{attribute 'pack_mode' := '0'}
TYPE ST_PLCOutputs :
STRUCT
	Q0: BYTE;
	Q1: BYTE;
	Q2: BYTE;
	Q3: BYTE;
	Q4: BYTE;
	Q5: BYTE;
	Q6: BYTE;
	Q7: BYTE;
	Q8: BYTE;
	Q9: BYTE;
	Q10: BYTE;
	Q11: BYTE;
	Q12: BYTE;
	Q13: BYTE;
	Q14: BYTE;
	Q15: BYTE;
	Q16: BYTE;
	Q17: BYTE;
	Q18: BYTE;
	Q19: BYTE;
	Q20: BYTE;
	Q21: BYTE;
	Q22: BYTE;
	Q23: BYTE;
	Q24: BYTE;
	Q25: BYTE;
	Q26: BYTE;
	Q27: BYTE;
	Q28: BYTE;
	Q29: BYTE;
	Q30: BYTE;
	Q31: BYTE;
	Q32: BYTE;
	Q33: BYTE;
	Q34: BYTE;
	Q35: BYTE;
	Q36: BYTE;
	Q37: BYTE;
	Q38: BYTE;
	Q39: BYTE;
	Q40: BYTE;
	Q41: BYTE;
	Q42: BYTE;
	Q43: BYTE;
	Q44: BYTE;
	Q45: BYTE;
	Q46: BYTE;
	Q47: BYTE;
	Q48: BYTE;
	Q49: BYTE;
	Q50: BYTE;
	Q51: BYTE;
	Q52: BYTE;
	Q53: BYTE;
	Q54: BYTE;
	Q55: BYTE;
	Q56: BYTE;
	Q57: BYTE;
	Q58: BYTE;
	Q59: BYTE;
	Q60: BYTE;
	Q61: BYTE;
	Q62: BYTE;
	Q63: BYTE;
	Q64: BYTE;
	Q65: BYTE;
	Q66: BYTE;
	Q67: BYTE;
	Q68: BYTE;
	Q69: BYTE;
	Q70: BYTE;
	Q71: BYTE;
	Q72: BYTE;
	Q73: BYTE;
	Q74: BYTE;
	Q75: BYTE;
	Q76: BYTE;
	Q77: BYTE;
	Q78: BYTE;
	Q79: BYTE;
	Q80: BYTE;
	Q81: BYTE;
	Q82: BYTE;
	Q83: BYTE;
	Q84: BYTE;
	Q85: BYTE;
	Q86: BYTE;
	Q87: BYTE;
	Q88: BYTE;
	Q89: BYTE;
	Q90: BYTE;
	Q91: BYTE;
	Q92: BYTE;
	Q93: BYTE;
	Q94: BYTE;
	Q95: BYTE;
	Q96: BYTE;
	Q97: BYTE;
	Q98: BYTE;
	Q99: BYTE;
	Q100: BYTE;
	Q101: BYTE;
	Q102: BYTE;
	Q103: BYTE;
	Q104: BYTE;
	Q105: BYTE;
	Q106: BYTE;
	Q107: BYTE;
	Q108: BYTE;
	Q109: BYTE;
	Q110: BYTE;
	Q111: BYTE;
	Q112: BYTE;
	Q113: BYTE;
	Q114: BYTE;
	Q115: BYTE;
	Q116: BYTE;
	Q117: BYTE;
	Q118: BYTE;
	Q119: BYTE;
	Q120: BYTE;
	Q121: BYTE;
	Q122: BYTE;
	Q123: BYTE;
	Q124: BYTE;
	Q125: BYTE;
	Q126: BYTE;
	Q127: BYTE;
	Q128: BYTE;
	Q129: BYTE;
	Q130: BYTE;
	Q131: BYTE;
	Q132: BYTE;
	Q133: BYTE;
	Q134: BYTE;
	Q135: BYTE;
	Q136: BYTE;
	Q137: BYTE;
	Q138: BYTE;
	Q139: BYTE;
	Q140: BYTE;
	Q141: BYTE;
	Q142: BYTE;
	Q143: BYTE;
	Q144: BYTE;
	Q145: BYTE;
	Q146: BYTE;
	Q147: BYTE;
	Q148: BYTE;
	Q149: BYTE;
	Q150: BYTE;
	Q151: BYTE;
	Q152: BYTE;
	Q153: BYTE;
	Q154: BYTE;
	Q155: BYTE;
	Q156: BYTE;
	Q157: BYTE;
	Q158: BYTE;
	Q159: BYTE;
	Q160: BYTE;
	Q161: BYTE;
	Q162: BYTE;
	Q163: BYTE;
	Q164: BYTE;
	Q165: BYTE;
	Q166: BYTE;
	Q167: BYTE;
	Q168: BYTE;
	Q169: BYTE;
	Q170: BYTE;
	Q171: BYTE;
	Q172: BYTE;
	Q173: BYTE;
	Q174: BYTE;
	Q175: BYTE;
	Q176: BYTE;
	Q177: BYTE;
	Q178: BYTE;
	Q179: BYTE;
	Q180: BYTE;
	Q181: BYTE;
	Q182: BYTE;
	Q183: BYTE;
	Q184: BYTE;
	Q185: BYTE;
	Q186: BYTE;
	Q187: BYTE;
	Q188: BYTE;
	Q189: BYTE;
	Q190: BYTE;
	Q191: BYTE;
	Q192: BYTE;
	Q193: BYTE;
	Q194: BYTE;
	Q195: BYTE;
	Q196: BYTE;
	Q197: BYTE;
	Q198: BYTE;
	Q199: BYTE;
	Q200: BYTE;
	Q201: BYTE;
	Q202: BYTE;
	Q203: BYTE;
	Q204: BYTE;
	Q205: BYTE;
	Q206: BYTE;
	Q207: BYTE;
	Q208: BYTE;
	Q209: BYTE;
	Q210: BYTE;
	Q211: BYTE;
	Q212: BYTE;
	Q213: BYTE;
	Q214: BYTE;
	Q215: BYTE;
	Q216: BYTE;
	Q217: BYTE;
	Q218: BYTE;
	Q219: BYTE;
	Q220: BYTE;
	Q221: BYTE;
	Q222: BYTE;
	Q223: BYTE;
	Q224: BYTE;
	Q225: BYTE;
	Q226: BYTE;
	Q227: BYTE;
	Q228: BYTE;
	Q229: BYTE;
	Q230: BYTE;
	Q231: BYTE;
	Q232: BYTE;
	Q233: BYTE;
	Q234: BYTE;
	Q235: BYTE;
	Q236: BYTE;
	Q237: BYTE;
	Q238: BYTE;
	Q239: BYTE;
	Q240: BYTE;
	Q241: BYTE;
	Q242: BYTE;
	Q243: BYTE;
	Q244: BYTE;
	Q245: BYTE;
	Q246: BYTE;
	Q247: BYTE;
	Q248: BYTE;
	Q249: BYTE;
	Q250: BYTE;
	Q251: BYTE;
	Q252: BYTE;
	Q253: BYTE;
	Q254: BYTE;
	Q255: BYTE;
	Q256: BYTE;
	Q257: BYTE;
	Q258: BYTE;
	Q259: BYTE;
	Q260: BYTE;
	Q261: BYTE;
	Q262: BYTE;
	Q263: BYTE;
	Q264: BYTE;
	Q265: BYTE;
	Q266: BYTE;
	Q267: BYTE;
	Q268: BYTE;
	Q269: BYTE;
	Q270: BYTE;
	Q271: BYTE;
	Q272: BYTE;
	Q273: BYTE;
	Q274: BYTE;
	Q275: BYTE;
	Q276: BYTE;
	Q277: BYTE;
	Q278: BYTE;
	Q279: BYTE;
	Q280: BYTE;
	Q281: BYTE;
	Q282: BYTE;
	Q283: BYTE;
	Q284: BYTE;
	Q285: BYTE;
	Q286: BYTE;
	Q287: BYTE;
	Q288: BYTE;
	Q289: BYTE;
	Q290: BYTE;
	Q291: BYTE;
	Q292: BYTE;
	Q293: BYTE;
	Q294: BYTE;
	Q295: BYTE;
	Q296: BYTE;
	Q297: BYTE;
	Q298: BYTE;
	Q299: BYTE;
	Q300: BYTE;
	Q301: BYTE;
	Q302: BYTE;
	Q303: BYTE;
	Q304: BYTE;
	Q305: BYTE;
	Q306: BYTE;
	Q307: BYTE;
	Q308: BYTE;
	Q309: BYTE;
	Q310: BYTE;
	Q311: BYTE;
	Q312: BYTE;
	Q313: BYTE;
	Q314: BYTE;
	Q315: BYTE;
	Q316: BYTE;
	Q317: BYTE;
	Q318: BYTE;
	Q319: BYTE;
	Q320: BYTE;
	Q321: BYTE;
	Q322: BYTE;
	Q323: BYTE;
	Q324: BYTE;
	Q325: BYTE;
	Q326: BYTE;
	Q327: BYTE;
	Q328: BYTE;
	Q329: BYTE;
	Q330: BYTE;
	Q331: BYTE;
	Q332: BYTE;
	Q333: BYTE;
	Q334: BYTE;
	Q335: BYTE;
	Q336: BYTE;
	Q337: BYTE;
	Q338: BYTE;
	Q339: BYTE;
	Q340: BYTE;
	Q341: BYTE;
	Q342: BYTE;
	Q343: BYTE;
	Q344: BYTE;
	Q345: BYTE;
	Q346: BYTE;
	Q347: BYTE;
	Q348: BYTE;
	Q349: BYTE;
	Q350: BYTE;
	Q351: BYTE;
	Q352: BYTE;
	Q353: BYTE;
	Q354: BYTE;
	Q355: BYTE;
	Q356: BYTE;
	Q357: BYTE;
	Q358: BYTE;
	Q359: BYTE;
	Q360: BYTE;
	Q361: BYTE;
	Q362: BYTE;
	Q363: BYTE;
	Q364: BYTE;
	Q365: BYTE;
	Q366: BYTE;
	Q367: BYTE;
	Q368: BYTE;
	Q369: BYTE;
	Q370: BYTE;
	Q371: BYTE;
	Q372: BYTE;
	Q373: BYTE;
	Q374: BYTE;
	Q375: BYTE;
	Q376: BYTE;
	Q377: BYTE;
	Q378: BYTE;
	Q379: BYTE;
	Q380: BYTE;
	Q381: BYTE;
	Q382: BYTE;
	Q383: BYTE;
	Q384: BYTE;
	Q385: BYTE;
	Q386: BYTE;
	Q387: BYTE;
	Q388: BYTE;
	Q389: BYTE;
	Q390: BYTE;
	Q391: BYTE;
	Q392: BYTE;
	Q393: BYTE;
	Q394: BYTE;
	Q395: BYTE;
	Q396: BYTE;
	Q397: BYTE;
	Q398: BYTE;
	Q399: BYTE;
	Q400: BYTE;
	Q401: BYTE;
	Q402: BYTE;
	Q403: BYTE;
	Q404: BYTE;
	Q405: BYTE;
	Q406: BYTE;
	Q407: BYTE;
	Q408: BYTE;
	Q409: BYTE;
	Q410: BYTE;
	Q411: BYTE;
	Q412: BYTE;
	Q413: BYTE;
	Q414: BYTE;
	Q415: BYTE;
	Q416: BYTE;
	Q417: BYTE;
	Q418: BYTE;
	Q419: BYTE;
	Q420: BYTE;
	Q421: BYTE;
	Q422: BYTE;
	Q423: BYTE;
	Q424: BYTE;
	Q425: BYTE;
	Q426: BYTE;
	Q427: BYTE;
	Q428: BYTE;
	Q429: BYTE;
	Q430: BYTE;
	Q431: BYTE;
	Q432: BYTE;
	Q433: BYTE;
	Q434: BYTE;
	Q435: BYTE;
	Q436: BYTE;
	Q437: BYTE;
	Q438: BYTE;
	Q439: BYTE;
	Q440: BYTE;
	Q441: BYTE;
	Q442: BYTE;
	Q443: BYTE;
	Q444: BYTE;
	Q445: BYTE;
	Q446: BYTE;
	Q447: BYTE;
	Q448: BYTE;
	Q449: BYTE;
	Q450: BYTE;
	Q451: BYTE;
	Q452: BYTE;
	Q453: BYTE;
	Q454: BYTE;
	Q455: BYTE;
	Q456: BYTE;
	Q457: BYTE;
	Q458: BYTE;
	Q459: BYTE;
	Q460: BYTE;
	Q461: BYTE;
	Q462: BYTE;
	Q463: BYTE;
	Q464: BYTE;
	Q465: BYTE;
	Q466: BYTE;
	Q467: BYTE;
	Q468: BYTE;
	Q469: BYTE;
	Q470: BYTE;
	Q471: BYTE;
	Q472: BYTE;
	Q473: BYTE;
	Q474: BYTE;
	Q475: BYTE;
	Q476: BYTE;
	Q477: BYTE;
	Q478: BYTE;
	Q479: BYTE;
	Q480: BYTE;
	Q481: BYTE;
	Q482: BYTE;
	Q483: BYTE;
	Q484: BYTE;
	Q485: BYTE;
	Q486: BYTE;
	Q487: BYTE;
	Q488: BYTE;
	Q489: BYTE;
	Q490: BYTE;
	Q491: BYTE;
	Q492: BYTE;
	Q493: BYTE;
	Q494: BYTE;
	Q495: BYTE;
	Q496: BYTE;
	Q497: BYTE;
	Q498: BYTE;
	Q499: BYTE;
	Q500: BYTE;
	Q501: BYTE;
	Q502: BYTE;
	Q503: BYTE;
	Q504: BYTE;
	Q505: BYTE;
	Q506: BYTE;
	Q507: BYTE;
	Q508: BYTE;
	Q509: BYTE;
	Q510: BYTE;
	Q511: BYTE;
	Q512: BYTE;
	Q513: BYTE;
	Q514: BYTE;
	Q515: BYTE;
	Q516: BYTE;
	Q517: BYTE;
	Q518: BYTE;
	Q519: BYTE;
	Q520: BYTE;
	Q521: BYTE;
	Q522: BYTE;
	Q523: BYTE;
	Q524: BYTE;
	Q525: BYTE;
	Q526: BYTE;
	Q527: BYTE;
	Q528: BYTE;
	Q529: BYTE;
	Q530: BYTE;
	Q531: BYTE;
	Q532: BYTE;
	Q533: BYTE;
	Q534: BYTE;
	Q535: BYTE;
	Q536: BYTE;
	Q537: BYTE;
	Q538: BYTE;
	Q539: BYTE;
	Q540: BYTE;
	Q541: BYTE;
	Q542: BYTE;
	Q543: BYTE;
	Q544: BYTE;
	Q545: BYTE;
	Q546: BYTE;
	Q547: BYTE;
	Q548: BYTE;
	Q549: BYTE;
	Q550: BYTE;
	Q551: BYTE;
	Q552: BYTE;
	Q553: BYTE;
	Q554: BYTE;
	Q555: BYTE;
	Q556: BYTE;
	Q557: BYTE;
	Q558: BYTE;
	Q559: BYTE;
	Q560: BYTE;
	Q561: BYTE;
	Q562: BYTE;
	Q563: BYTE;
	Q564: BYTE;
	Q565: BYTE;
	Q566: BYTE;
	Q567: BYTE;
	Q568: BYTE;
	Q569: BYTE;
	Q570: BYTE;
	Q571: BYTE;
	Q572: BYTE;
	Q573: BYTE;
	Q574: BYTE;
	Q575: BYTE;
	Q576: BYTE;
	Q577: BYTE;
	Q578: BYTE;
	Q579: BYTE;
	Q580: BYTE;
	Q581: BYTE;
	Q582: BYTE;
	Q583: BYTE;
	Q584: BYTE;
	Q585: BYTE;
	Q586: BYTE;
	Q587: BYTE;
	Q588: BYTE;
	Q589: BYTE;
	Q590: BYTE;
	Q591: BYTE;
	Q592: BYTE;
	Q593: BYTE;
	Q594: BYTE;
	Q595: BYTE;
	Q596: BYTE;
	Q597: BYTE;
	Q598: BYTE;
	Q599: BYTE;
	Q600: BYTE;
	Q601: BYTE;
	Q602: BYTE;
	Q603: BYTE;
	Q604: BYTE;
	Q605: BYTE;
	Q606: BYTE;
	Q607: BYTE;
	Q608: BYTE;
	Q609: BYTE;
	Q610: BYTE;
	Q611: BYTE;
	Q612: BYTE;
	Q613: BYTE;
	Q614: BYTE;
	Q615: BYTE;
	Q616: BYTE;
	Q617: BYTE;
	Q618: BYTE;
	Q619: BYTE;
	Q620: BYTE;
	Q621: BYTE;
	Q622: BYTE;
	Q623: BYTE;
	Q624: BYTE;
	Q625: BYTE;
	Q626: BYTE;
	Q627: BYTE;
	Q628: BYTE;
	Q629: BYTE;
	Q630: BYTE;
	Q631: BYTE;
	Q632: BYTE;
	Q633: BYTE;
	Q634: BYTE;
	Q635: BYTE;
	Q636: BYTE;
	Q637: BYTE;
	Q638: BYTE;
	Q639: BYTE;
	Q640: BYTE;
	Q641: BYTE;
	Q642: BYTE;
	Q643: BYTE;
	Q644: BYTE;
	Q645: BYTE;
	Q646: BYTE;
	Q647: BYTE;
	Q648: BYTE;
	Q649: BYTE;
	Q650: BYTE;
	Q651: BYTE;
	Q652: BYTE;
	Q653: BYTE;
	Q654: BYTE;
	Q655: BYTE;
	Q656: BYTE;
	Q657: BYTE;
	Q658: BYTE;
	Q659: BYTE;
	Q660: BYTE;
	Q661: BYTE;
	Q662: BYTE;
	Q663: BYTE;
	Q664: BYTE;
	Q665: BYTE;
	Q666: BYTE;
	Q667: BYTE;
	Q668: BYTE;
	Q669: BYTE;
	Q670: BYTE;
	Q671: BYTE;
	Q672: BYTE;
	Q673: BYTE;
	Q674: BYTE;
	Q675: BYTE;
	Q676: BYTE;
	Q677: BYTE;
	Q678: BYTE;
	Q679: BYTE;
	Q680: BYTE;
	Q681: BYTE;
	Q682: BYTE;
	Q683: BYTE;
	Q684: BYTE;
	Q685: BYTE;
	Q686: BYTE;
	Q687: BYTE;
	Q688: BYTE;
	Q689: BYTE;
	Q690: BYTE;
	Q691: BYTE;
	Q692: BYTE;
	Q693: BYTE;
	Q694: BYTE;
	Q695: BYTE;
	Q696: BYTE;
	Q697: BYTE;
	Q698: BYTE;
	Q699: BYTE;
	Q700: BYTE;
	Q701: BYTE;
	Q702: BYTE;
	Q703: BYTE;
	Q704: BYTE;
	Q705: BYTE;
	Q706: BYTE;
	Q707: BYTE;
	Q708: BYTE;
	Q709: BYTE;
	Q710: BYTE;
	Q711: BYTE;
	Q712: BYTE;
	Q713: BYTE;
	Q714: BYTE;
	Q715: BYTE;
	Q716: BYTE;
	Q717: BYTE;
	Q718: BYTE;
	Q719: BYTE;
	Q720: BYTE;
	Q721: BYTE;
	Q722: BYTE;
	Q723: BYTE;
	Q724: BYTE;
	Q725: BYTE;
	Q726: BYTE;
	Q727: BYTE;
	Q728: BYTE;
	Q729: BYTE;
	Q730: BYTE;
	Q731: BYTE;
	Q732: BYTE;
	Q733: BYTE;
	Q734: BYTE;
	Q735: BYTE;
	Q736: BYTE;
	Q737: BYTE;
	Q738: BYTE;
	Q739: BYTE;
	Q740: BYTE;
	Q741: BYTE;
	Q742: BYTE;
	Q743: BYTE;
	Q744: BYTE;
	Q745: BYTE;
	Q746: BYTE;
	Q747: BYTE;
	Q748: BYTE;
	Q749: BYTE;
	Q750: BYTE;
	Q751: BYTE;
	Q752: BYTE;
	Q753: BYTE;
	Q754: BYTE;
	Q755: BYTE;
	Q756: BYTE;
	Q757: BYTE;
	Q758: BYTE;
	Q759: BYTE;
	Q760: BYTE;
	Q761: BYTE;
	Q762: BYTE;
	Q763: BYTE;
	Q764: BYTE;
	Q765: BYTE;
	Q766: BYTE;
	Q767: BYTE;
	Q768: BYTE;
	Q769: BYTE;
	Q770: BYTE;
	Q771: BYTE;
	Q772: BYTE;
	Q773: BYTE;
	Q774: BYTE;
	Q775: BYTE;
	Q776: BYTE;
	Q777: BYTE;
	Q778: BYTE;
	Q779: BYTE;
	Q780: BYTE;
	Q781: BYTE;
	Q782: BYTE;
	Q783: BYTE;
	Q784: BYTE;
	Q785: BYTE;
	Q786: BYTE;
	Q787: BYTE;
	Q788: BYTE;
	Q789: BYTE;
	Q790: BYTE;
	Q791: BYTE;
	Q792: BYTE;
	Q793: BYTE;
	Q794: BYTE;
	Q795: BYTE;
	Q796: BYTE;
	Q797: BYTE;
	Q798: BYTE;
	Q799: BYTE;
	Q800: BYTE;
	Q801: BYTE;
	Q802: BYTE;
	Q803: BYTE;
	Q804: BYTE;
	Q805: BYTE;
	Q806: BYTE;
	Q807: BYTE;
	Q808: BYTE;
	Q809: BYTE;
	Q810: BYTE;
	Q811: BYTE;
	Q812: BYTE;
	Q813: BYTE;
	Q814: BYTE;
	Q815: BYTE;
	Q816: BYTE;
	Q817: BYTE;
	Q818: BYTE;
	Q819: BYTE;
	Q820: BYTE;
	Q821: BYTE;
	Q822: BYTE;
	Q823: BYTE;
	Q824: BYTE;
	Q825: BYTE;
	Q826: BYTE;
	Q827: BYTE;
	Q828: BYTE;
	Q829: BYTE;
	Q830: BYTE;
	Q831: BYTE;
	Q832: BYTE;
	Q833: BYTE;
	Q834: BYTE;
	Q835: BYTE;
	Q836: BYTE;
	Q837: BYTE;
	Q838: BYTE;
	Q839: BYTE;
	Q840: BYTE;
	Q841: BYTE;
	Q842: BYTE;
	Q843: BYTE;
	Q844: BYTE;
	Q845: BYTE;
	Q846: BYTE;
	Q847: BYTE;
	Q848: BYTE;
	Q849: BYTE;
	Q850: BYTE;
	Q851: BYTE;
	Q852: BYTE;
	Q853: BYTE;
	Q854: BYTE;
	Q855: BYTE;
	Q856: BYTE;
	Q857: BYTE;
	Q858: BYTE;
	Q859: BYTE;
	Q860: BYTE;
	Q861: BYTE;
	Q862: BYTE;
	Q863: BYTE;
	Q864: BYTE;
	Q865: BYTE;
	Q866: BYTE;
	Q867: BYTE;
	Q868: BYTE;
	Q869: BYTE;
	Q870: BYTE;
	Q871: BYTE;
	Q872: BYTE;
	Q873: BYTE;
	Q874: BYTE;
	Q875: BYTE;
	Q876: BYTE;
	Q877: BYTE;
	Q878: BYTE;
	Q879: BYTE;
	Q880: BYTE;
	Q881: BYTE;
	Q882: BYTE;
	Q883: BYTE;
	Q884: BYTE;
	Q885: BYTE;
	Q886: BYTE;
	Q887: BYTE;
	Q888: BYTE;
	Q889: BYTE;
	Q890: BYTE;
	Q891: BYTE;
	Q892: BYTE;
	Q893: BYTE;
	Q894: BYTE;
	Q895: BYTE;
	Q896: BYTE;
	Q897: BYTE;
	Q898: BYTE;
	Q899: BYTE;
	Q900: BYTE;
	Q901: BYTE;
	Q902: BYTE;
	Q903: BYTE;
	Q904: BYTE;
	Q905: BYTE;
	Q906: BYTE;
	Q907: BYTE;
	Q908: BYTE;
	Q909: BYTE;
	Q910: BYTE;
	Q911: BYTE;
	Q912: BYTE;
	Q913: BYTE;
	Q914: BYTE;
	Q915: BYTE;
	Q916: BYTE;
	Q917: BYTE;
	Q918: BYTE;
	Q919: BYTE;
	Q920: BYTE;
	Q921: BYTE;
	Q922: BYTE;
	Q923: BYTE;
	Q924: BYTE;
	Q925: BYTE;
	Q926: BYTE;
	Q927: BYTE;
	Q928: BYTE;
	Q929: BYTE;
	Q930: BYTE;
	Q931: BYTE;
	Q932: BYTE;
	Q933: BYTE;
	Q934: BYTE;
	Q935: BYTE;
	Q936: BYTE;
	Q937: BYTE;
	Q938: BYTE;
	Q939: BYTE;
	Q940: BYTE;
	Q941: BYTE;
	Q942: BYTE;
	Q943: BYTE;
	Q944: BYTE;
	Q945: BYTE;
	Q946: BYTE;
	Q947: BYTE;
	Q948: BYTE;
	Q949: BYTE;
	Q950: BYTE;
	Q951: BYTE;
	Q952: BYTE;
	Q953: BYTE;
	Q954: BYTE;
	Q955: BYTE;
	Q956: BYTE;
	Q957: BYTE;
	Q958: BYTE;
	Q959: BYTE;
	Q960: BYTE;
	Q961: BYTE;
	Q962: BYTE;
	Q963: BYTE;
	Q964: BYTE;
	Q965: BYTE;
	Q966: BYTE;
	Q967: BYTE;
	Q968: BYTE;
	Q969: BYTE;
	Q970: BYTE;
	Q971: BYTE;
	Q972: BYTE;
	Q973: BYTE;
	Q974: BYTE;
	Q975: BYTE;
	Q976: BYTE;
	Q977: BYTE;
	Q978: BYTE;
	Q979: BYTE;
	Q980: BYTE;
	Q981: BYTE;
	Q982: BYTE;
	Q983: BYTE;
	Q984: BYTE;
	Q985: BYTE;
	Q986: BYTE;
	Q987: BYTE;
	Q988: BYTE;
	Q989: BYTE;
	Q990: BYTE;
	Q991: BYTE;
	Q992: BYTE;
	Q993: BYTE;
	Q994: BYTE;
	Q995: BYTE;
	Q996: BYTE;
	Q997: BYTE;
	Q998: BYTE;
	Q999: BYTE;
	Q1000: BYTE;
	Q1001: BYTE;
	Q1002: BYTE;
	Q1003: BYTE;
	Q1004: BYTE;
	Q1005: BYTE;
	Q1006: BYTE;
	Q1007: BYTE;
	Q1008: BYTE;
	Q1009: BYTE;
	Q1010: BYTE;
	Q1011: BYTE;
	Q1012: BYTE;
	Q1013: BYTE;
	Q1014: BYTE;
	Q1015: BYTE;
	Q1016: BYTE;
	Q1017: BYTE;
	Q1018: BYTE;
	Q1019: BYTE;
	Q1020: BYTE;
	Q1021: BYTE;
	Q1022: BYTE;
	Q1023: BYTE;
END_STRUCT
END_TYPE

(* stored: Version 1.1.0.1, ProductVersion 3.1.4026.18
   DUT ST_PLCOutputs: Id {becafd5c-cb0b-43ea-b755-87130a177863} *)
